// TIA Portal V19 export
FUNCTION_BLOCK "MainSafety"   // FB900, F_LAD
{ S7_Optimized_Access := 'TRUE' }
// stored: AutoNumber false
BEGIN

REGION Network 1: Read input safety from left robot
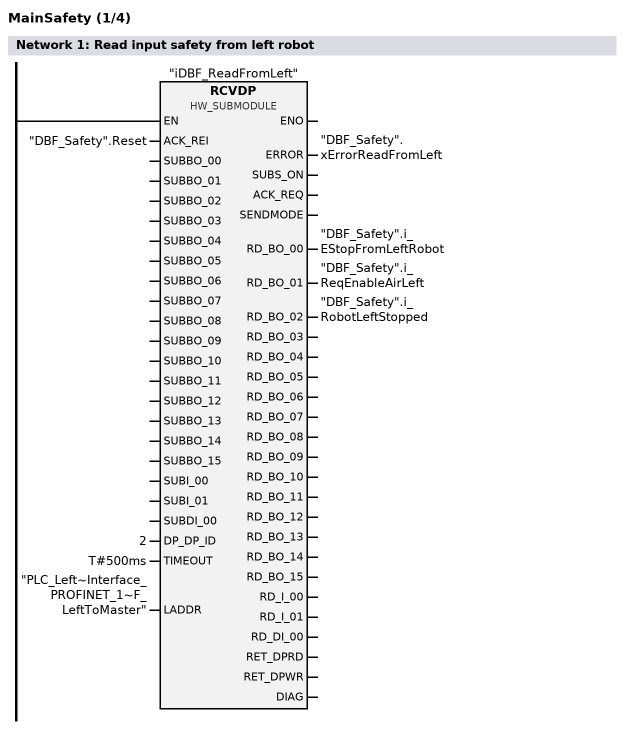
   RUNG wire#powerrail
      { S7_Templates := "laddr_type := HW_SUBMODULE" } "iDBF_ReadFromLeft".RCVDP(ACK_REI := "DBF_Safety".Reset, SUBBO_00 :=, SUBBO_01 :=, SUBBO_02 :=, SUBBO_03 :=, SUBBO_04 :=, SUBBO_05 :=, SUBBO_06 :=, SUBBO_07 :=, SUBBO_08 :=, SUBBO_09 :=, SUBBO_10 :=, SUBBO_11 :=, SUBBO_12 :=, SUBBO_13 :=, SUBBO_14 :=, SUBBO_15 :=, SUBI_00 :=, SUBI_01 :=, SUBDI_00 :=, DP_DP_ID := 2, TIMEOUT := T#500ms, LADDR := "PLC_Left~Interface_PROFINET_1~F_LeftToMaster", ERROR => "DBF_Safety".xErrorReadFromLeft, SUBS_ON =>, ACK_REQ =>, SENDMODE =>, RD_BO_00 => "DBF_Safety".i_EStopFromLeftRobot, RD_BO_01 => "DBF_Safety".i_ReqEnableAirLeft, RD_BO_02 => "DBF_Safety".i_RobotLeftStopped, RD_BO_03 =>, RD_BO_04 =>, RD_BO_05 =>, RD_BO_06 =>, RD_BO_07 =>, RD_BO_08 =>, RD_BO_09 =>, RD_BO_10 =>, RD_BO_11 =>, RD_BO_12 =>, RD_BO_13 =>, RD_BO_14 =>, RD_BO_15 =>, RD_I_00 =>, RD_I_01 =>, RD_DI_00 =>, RET_DPRD =>, RET_DPWR =>, DIAG =>)
   END_RUNG
   // the same network as SCL:
   "iDBF_ReadFromLeft"(ACK_REI := "DBF_Safety".Reset,   // RCVDP
                       DP_DP_ID := 2,
                       TIMEOUT := T#500ms,
                       LADDR := "PLC_Left~Interface_PROFINET_1~F_LeftToMaster",
                       ERROR => "DBF_Safety".xErrorReadFromLeft,
                       RD_BO_00 => "DBF_Safety".i_EStopFromLeftRobot,
                       RD_BO_01 => "DBF_Safety".i_ReqEnableAirLeft,
                       RD_BO_02 => "DBF_Safety".i_RobotLeftStopped);
END_REGION

REGION Network 2: Read input safety from right robot
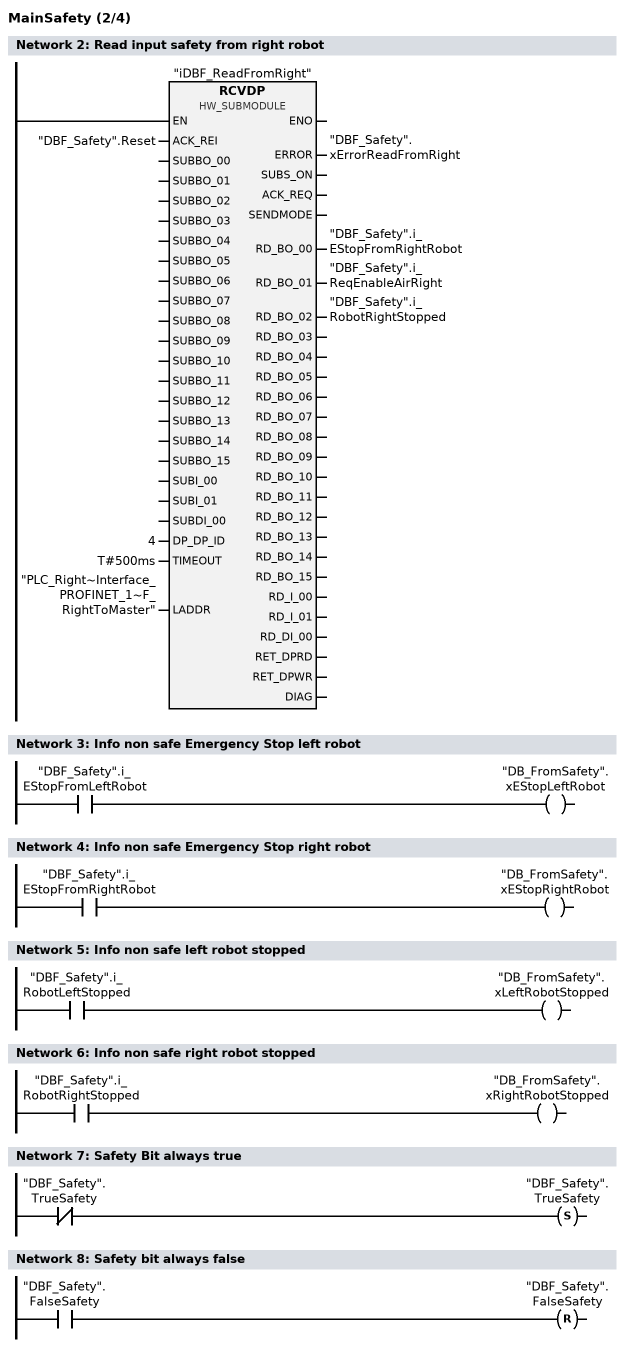
   RUNG wire#powerrail
      { S7_Templates := "laddr_type := HW_SUBMODULE" } "iDBF_ReadFromRight".RCVDP(ACK_REI := "DBF_Safety".Reset, SUBBO_00 :=, SUBBO_01 :=, SUBBO_02 :=, SUBBO_03 :=, SUBBO_04 :=, SUBBO_05 :=, SUBBO_06 :=, SUBBO_07 :=, SUBBO_08 :=, SUBBO_09 :=, SUBBO_10 :=, SUBBO_11 :=, SUBBO_12 :=, SUBBO_13 :=, SUBBO_14 :=, SUBBO_15 :=, SUBI_00 :=, SUBI_01 :=, SUBDI_00 :=, DP_DP_ID := 4, TIMEOUT := T#500ms, LADDR := "PLC_Right~Interface_PROFINET_1~F_RightToMaster", ERROR => "DBF_Safety".xErrorReadFromRight, SUBS_ON =>, ACK_REQ =>, SENDMODE =>, RD_BO_00 => "DBF_Safety".i_EStopFromRightRobot, RD_BO_01 => "DBF_Safety".i_ReqEnableAirRight, RD_BO_02 => "DBF_Safety".i_RobotRightStopped, RD_BO_03 =>, RD_BO_04 =>, RD_BO_05 =>, RD_BO_06 =>, RD_BO_07 =>, RD_BO_08 =>, RD_BO_09 =>, RD_BO_10 =>, RD_BO_11 =>, RD_BO_12 =>, RD_BO_13 =>, RD_BO_14 =>, RD_BO_15 =>, RD_I_00 =>, RD_I_01 =>, RD_DI_00 =>, RET_DPRD =>, RET_DPWR =>, DIAG =>)
   END_RUNG
   // the same network as SCL:
   "iDBF_ReadFromRight"(ACK_REI := "DBF_Safety".Reset,   // RCVDP
                        DP_DP_ID := 4,
                        TIMEOUT := T#500ms,
                        LADDR := "PLC_Right~Interface_PROFINET_1~F_RightToMaster",
                        ERROR => "DBF_Safety".xErrorReadFromRight,
                        RD_BO_00 => "DBF_Safety".i_EStopFromRightRobot,
                        RD_BO_01 => "DBF_Safety".i_ReqEnableAirRight,
                        RD_BO_02 => "DBF_Safety".i_RobotRightStopped);
END_REGION

REGION Network 3: Info non safe Emergency Stop left robot
   RUNG wire#powerrail
      Contact( "DBF_Safety".i_EStopFromLeftRobot )
      Coil( "DB_FromSafety".xEStopLeftRobot )
   END_RUNG
   // the same network as SCL:
   "DB_FromSafety".xEStopLeftRobot := "DBF_Safety".i_EStopFromLeftRobot;
END_REGION

REGION Network 4: Info non safe Emergency Stop right robot
   RUNG wire#powerrail
      Contact( "DBF_Safety".i_EStopFromRightRobot )
      Coil( "DB_FromSafety".xEStopRightRobot )
   END_RUNG
   // the same network as SCL:
   "DB_FromSafety".xEStopRightRobot := "DBF_Safety".i_EStopFromRightRobot;
END_REGION

REGION Network 5: Info non safe left robot stopped
   RUNG wire#powerrail
      Contact( "DBF_Safety".i_RobotLeftStopped )
      Coil( "DB_FromSafety".xLeftRobotStopped )
   END_RUNG
   // the same network as SCL:
   "DB_FromSafety".xLeftRobotStopped := "DBF_Safety".i_RobotLeftStopped;
END_REGION

REGION Network 6: Info non safe right robot stopped
   RUNG wire#powerrail
      Contact( "DBF_Safety".i_RobotRightStopped )
      Coil( "DB_FromSafety".xRightRobotStopped )
   END_RUNG
   // the same network as SCL:
   "DB_FromSafety".xRightRobotStopped := "DBF_Safety".i_RobotRightStopped;
END_REGION

REGION Network 7: Safety Bit always true
   RUNG wire#powerrail
      I_Contact( "DBF_Safety".TrueSafety )
      S_Coil( "DBF_Safety".TrueSafety )
   END_RUNG
   // the same network as SCL:
   IF NOT "DBF_Safety".TrueSafety THEN "DBF_Safety".TrueSafety := TRUE; END_IF;
END_REGION

REGION Network 8: Safety bit always false
   RUNG wire#powerrail
      Contact( "DBF_Safety".FalseSafety )
      R_Coil( "DBF_Safety".FalseSafety )
   END_RUNG
   // the same network as SCL:
   IF "DBF_Safety".FalseSafety THEN "DBF_Safety".FalseSafety := FALSE; END_IF;
END_REGION

REGION Network 9: Safety reintegration function call
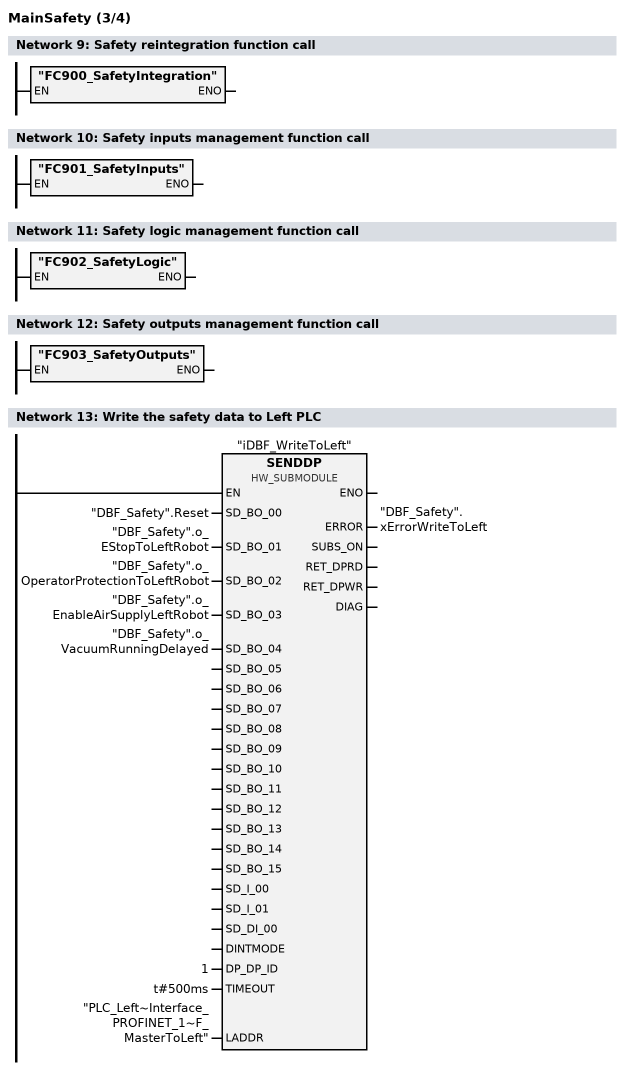
   RUNG wire#powerrail
      "FC900_SafetyIntegration"()
   END_RUNG
   // the same network as SCL:
   "FC900_SafetyIntegration"();
END_REGION

REGION Network 10: Safety inputs management function call
   RUNG wire#powerrail
      "FC901_SafetyInputs"()
   END_RUNG
   // the same network as SCL:
   "FC901_SafetyInputs"();
END_REGION

REGION Network 11: Safety logic management function call
   RUNG wire#powerrail
      "FC902_SafetyLogic"()
   END_RUNG
   // the same network as SCL:
   "FC902_SafetyLogic"();
END_REGION

REGION Network 12: Safety outputs management function call
   RUNG wire#powerrail
      "FC903_SafetyOutputs"()
   END_RUNG
   // the same network as SCL:
   "FC903_SafetyOutputs"();
END_REGION

REGION Network 13: Write the safety data to Left PLC
   RUNG wire#powerrail
      { S7_Templates := "laddr_type := HW_SUBMODULE" } "iDBF_WriteToLeft".SENDDP(SD_BO_00 := "DBF_Safety".Reset, SD_BO_01 := "DBF_Safety".o_EStopToLeftRobot, SD_BO_02 := "DBF_Safety".o_OperatorProtectionToLeftRobot, SD_BO_03 := "DBF_Safety".o_EnableAirSupplyLeftRobot, SD_BO_04 := "DBF_Safety".o_VacuumRunningDelayed, SD_BO_05 :=, SD_BO_06 :=, SD_BO_07 :=, SD_BO_08 :=, SD_BO_09 :=, SD_BO_10 :=, SD_BO_11 :=, SD_BO_12 :=, SD_BO_13 :=, SD_BO_14 :=, SD_BO_15 :=, SD_I_00 :=, SD_I_01 :=, SD_DI_00 :=, DINTMODE :=, DP_DP_ID := 1, TIMEOUT := t#500ms, LADDR := "PLC_Left~Interface_PROFINET_1~F_MasterToLeft", ERROR => "DBF_Safety".xErrorWriteToLeft, SUBS_ON =>, RET_DPRD =>, RET_DPWR =>, DIAG =>)
   END_RUNG
   // the same network as SCL:
   "iDBF_WriteToLeft"(SD_BO_00 := "DBF_Safety".Reset,   // SENDDP
                      SD_BO_01 := "DBF_Safety".o_EStopToLeftRobot,
                      SD_BO_02 := "DBF_Safety".o_OperatorProtectionToLeftRobot,
                      SD_BO_03 := "DBF_Safety".o_EnableAirSupplyLeftRobot,
                      SD_BO_04 := "DBF_Safety".o_VacuumRunningDelayed,
                      DP_DP_ID := 1,
                      TIMEOUT := t#500ms,
                      LADDR := "PLC_Left~Interface_PROFINET_1~F_MasterToLeft",
                      ERROR => "DBF_Safety".xErrorWriteToLeft);
END_REGION

REGION Network 14: Write the safety data to Right PLC
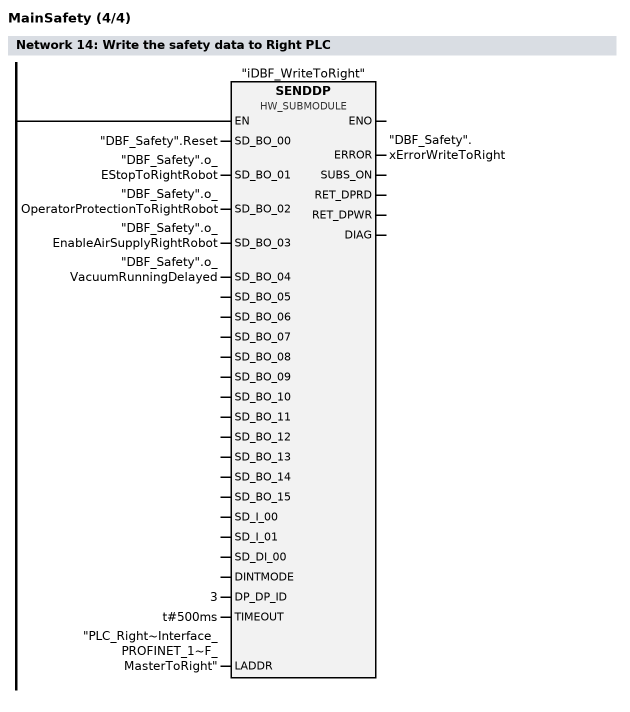
   RUNG wire#powerrail
      { S7_Templates := "laddr_type := HW_SUBMODULE" } "iDBF_WriteToRight".SENDDP(SD_BO_00 := "DBF_Safety".Reset, SD_BO_01 := "DBF_Safety".o_EStopToRightRobot, SD_BO_02 := "DBF_Safety".o_OperatorProtectionToRightRobot, SD_BO_03 := "DBF_Safety".o_EnableAirSupplyRightRobot, SD_BO_04 := "DBF_Safety".o_VacuumRunningDelayed, SD_BO_05 :=, SD_BO_06 :=, SD_BO_07 :=, SD_BO_08 :=, SD_BO_09 :=, SD_BO_10 :=, SD_BO_11 :=, SD_BO_12 :=, SD_BO_13 :=, SD_BO_14 :=, SD_BO_15 :=, SD_I_00 :=, SD_I_01 :=, SD_DI_00 :=, DINTMODE :=, DP_DP_ID := 3, TIMEOUT := t#500ms, LADDR := "PLC_Right~Interface_PROFINET_1~F_MasterToRight", ERROR => "DBF_Safety".xErrorWriteToRight, SUBS_ON =>, RET_DPRD =>, RET_DPWR =>, DIAG =>)
   END_RUNG
   // the same network as SCL:
   "iDBF_WriteToRight"(SD_BO_00 := "DBF_Safety".Reset,   // SENDDP
                       SD_BO_01 := "DBF_Safety".o_EStopToRightRobot,
                       SD_BO_02 := "DBF_Safety".o_OperatorProtectionToRightRobot,
                       SD_BO_03 := "DBF_Safety".o_EnableAirSupplyRightRobot,
                       SD_BO_04 := "DBF_Safety".o_VacuumRunningDelayed,
                       DP_DP_ID := 3,
                       TIMEOUT := t#500ms,
                       LADDR := "PLC_Right~Interface_PROFINET_1~F_MasterToRight",
                       ERROR => "DBF_Safety".xErrorWriteToRight);
END_REGION
END_FUNCTION_BLOCK
